{attribute addProperty BoxType "CX2040 EtherCAT slave-1b82-0016"}
{attribute addProperty Id "IO_InputsEMPTY_STRUCTURE000Device_Status_MappingAT %I*Device_Status_Mapping_AC515E2C1620IO_OutputsEMPTY_STRUCTURE000WcStateAT %I*WcState_98A4DF7520.250InfoDataAT %I*InfoData_275E3363128160"}
{attribute addProperty CRC "257024818"}
{attribute addProperty SizeInBites "146"}
{attribute addProperty SizeInBytes "18.25"}
TYPE CX2040_EtherCAT_slave_16898E41 :
STRUCT
	{attribute addProperty Name "IO_Inputs"}
	IO_Inputs : EMPTY_STRUCTURE;
	{attribute addProperty Name "Device_Status_Mapping"}
	Device_Status_Mapping : Device_Status_Mapping_AC515E2C;
	{attribute addProperty Name "IO_Outputs"}
	IO_Outputs : EMPTY_STRUCTURE;
	{attribute addProperty Name "WcState"}
	WcState : WcState_98A4DF75;
	{attribute addProperty Name "InfoData"}
	InfoData : InfoData_275E3363;
END_STRUCT
END_TYPE

(* stored: Version 1.2.0.0, ProductVersion 3.1.4024.9
   DUT CX2040_EtherCAT_slave_16898E41: Id {557f31ba-3cb5-469b-abc0-3e9196c3836a} *)
